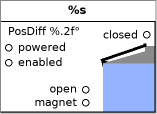
VISUALIZATION VISU_CoverPanelDetails  // 157x114
VAR_IN_OUT
    config : CoverPanelConfig;
	panel  : CoverPanel;
	widget : CoverPanelWidget;
    magnetEnabled : BOOL;
END_VAR
    Rectangle (0,21 155x91)
        p3450524324: widget.actualStatus.color.bg
    Polygon (101,60) (111,62) (103,68)
    Rectangle (0,0 155x20), "%s", text variable: config.name
    Rectangle (103,63 51x48)
    Polygon (103,63) (145,51) (145,46) (154,46) (154,63) (154,63)
    Polyline (101,60) (145,45) (145,45)
        p2858320360: widget.drawingAngle
    Ellipse (143,31 7x7), colour toggle: panel.statuses.apertureStatus.closed
    Rectangle (97,28 44x14), "closed"
    Rectangle (39,82 41x14), "open"
    Ellipse (82,86 7x7), colour toggle: panel.statuses.apertureStatus.open
    Ellipse (82,99 7x7), colour toggle: magnetEnabled
    Rectangle (29,95 51x15), "magnet"
    Rectangle (5,25 76x13), "PosDiff %.2f°", text variable: panel.parts.axis.axis_ref.NcToPlc.PosDiff
    Ellipse (5,59 7x7), colour toggle: panel.parts.axis.statuses.poweredStatus.enabled
    Rectangle (15,55 60x15), "enabled"
    Rectangle (15,40 55x15), "powered"
    Ellipse (5,44 7x7), colour toggle: panel.parts.motorRelay.digitalOutput
END_VISUALIZATION

(* stored: Version 1.1.0.1, ProductVersion 3.1.0.36
   Visu VISU_CoverPanelDetails: Id {fea757c9-da48-4708-84c8-dde3e124c884} *)
